/// This function block is a container for all axis objects that are used by this unit.
/// The parent of all objects can be directly transfered in their constructor (this is only relevant for equipment objects
/// that have to be managed (e.g. [DebouncedInput](xref:ZEquipment.DebouncedInput), [Light](xref:ZEquipment.Light), ...).
FUNCTION_BLOCK GearFieldbus EXTENDS GearContainer
VAR
END_VAR
VAR_INPUT

{attribute '__ZwPlcUnitEquipmentDeclaration__'} // Do not remove this attribute! It is used for code generation.
END_VAR

IF _isInitialized
THEN
  RETURN;
END_IF

{attribute '__ZwPlcUnitEquipmentImplementation__'} // Do not remove this attribute! It is used for code generation.

_isInitialized := TRUE;

END_FUNCTION_BLOCK

(* stored: Version 1.1.0.1
   POU GearFieldbus: Id {b6c54b4d-69c1-4f7c-818b-93d8c79271cd}, SpecialFunc None *)
